{attribute 'reflection'}
FUNCTION_BLOCK PUBLIC FB_DevAnalogInputScaled EXTENDS FB_DevAnalogInput
VAR_INPUT
END_VAR
VAR_OUTPUT
END_VAR
VAR
	nLimitMin		: INT := IBF_Utilities.GVL_FixedValues.nINTMINVALUE	; // Initial value is set to integer minimum value for use with normal def analog inputs 
	nLimitMax 		: INT := IBF_Utilities.GVL_FixedValues.nINTMAXVALUE	; // Initial value is set to integer minimum value for use with high def analog inputs
	fGainFactor 	: LREAL	:= 1	;
	nOfset			: INT	:= 0	;
END_VAR

SUPER^(refFbFault := refFbFault);

METHOD ExecSetFeedback : BOOL
VAR
	nCalibValue	: INT ; 
END_VAR
// Offset 
IF bCmdSimulate THEN 
	nCalibValue := fSimValue + nOfset ;
ELSE
	nCalibValue := inHwInput + nOfset ;
END_IF

fValue := INT_TO_LREAL(nCalibValue) / fGainFactor;

ExecSetFeedback := TRUE;
END_METHOD

METHOD PUBLIC SetScaling : BOOL 
VAR_INPUT
	fMaxValue	: LREAL ; 	// Maximum input value after scaling, e.g. 100%, 0 = no scaling (gain = hardware limit / fMaxValue)  
	fOfset		: LREAL ;	// offset value (fvalue = (gain * hwvalue) + fOfset)
END_VAR
// calculate gain 
IF fMaxValue =0 THEN 
	fGainFactor := 1 ;
ELSE 
	fGainFactor := nLimitMax / fMaxValue ;
END_IF

nOfset := LREAL_TO_INT(fOfset * fGainFactor) ;

SetScaling := TRUE;
END_METHOD

END_FUNCTION_BLOCK

(* stored: Version 1.1.0.1, ProductVersion 3.1.4024.11
   POU FB_DevAnalogInputScaled: Id {43638945-f4e4-0cff-025b-6c03ae4b4de9}, SpecialFunc None
   Method ExecSetFeedback: Id {6b8ba436-87f3-0e59-2933-34440dde902f}
   Method SetScaling: Id {ac76234a-a867-0b26-0f7d-98f1a69590d3} *)
